(* LS Electric XG5000 project: automatic Star-Delta *)
(* PLC LSPLC *)

PROGRAM NewProgram (* task: Scan Program *)
VAR
    delta AT %QX0.0.1 : BOOL;
    INST : TON;
    mc_c : BOOL;
    off AT %IX0.0.0 : BOOL;
    on AT %IX0.0.1 : BOOL;
    star AT %QX0.0.0 : BOOL;
END_VAR

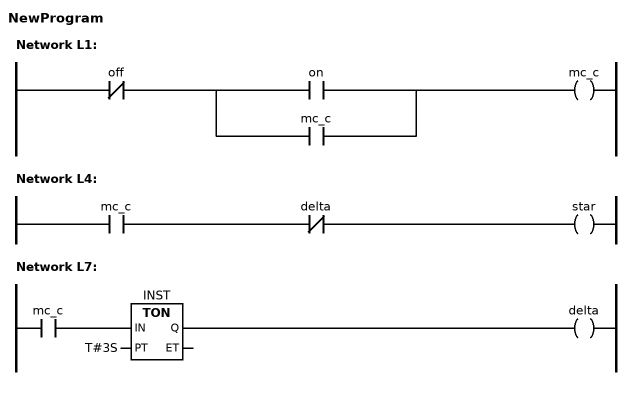
(* Rung L1 *)
mc_c := NOT off AND (on OR mc_c);
(* Rung L4 *)
star := mc_c AND NOT delta;
(* Rung L7 *)
INST(IN := mc_c, PT := T#3S);
delta := INST.Q;
END_PROGRAM